// TwinCAT 3 PLC project PLC1
// ProgramVersion: 3.1.4022.2
// libraries:
//   Tc2_IoFunctions, * (Beckhoff Automation GmbH)
//   Tc2_ModbusRTU, * (Beckhoff Automation GmbH)
//   Tc2_ModbusSrv, * (Beckhoff Automation GmbH)
//   Tc2_Standard, * (Beckhoff Automation GmbH)
//   Tc2_System, * (Beckhoff Automation GmbH)
//   Tc3_Module, * (Beckhoff Automation GmbH)
//   Tc3_PLCopen_OpcUa, * (Beckhoff Automation GmbH)
// project tree:
//   DUTs/ ATV212.TcDUT, ATV212RegAddress.TcDUT, GrundfosMagna3.TcDUT (not stored), GrundfosRegAddress.TcDUT (not stored)
//   GVLs/ GVL.TcGVL, HWVar.TcGVL (not stored), Scale.TcGVL
//   / ModbusComm.TcTTO (not stored), PlcTask.TcTTO (not stored)
//   POUs/ BackgroundComm.TcPOU (not stored), IOConversion.TcPOU (not stored), MAIN.TcPOU (not stored), ModbusCommunication.TcPOU

// ---- DUTs/ATV212.TcDUT
TYPE ATV212 :
STRUCT
	fOutputFrequencyStatus	: REAL;
	fOutputCurrentStatus	: REAL;
	fOutputVoltageStatus	: REAL;
	fMotorSpeedStatus		: REAL;
END_STRUCT
END_TYPE

// ---- DUTs/ATV212RegAddress.TcDUT
{attribute 'qualified_only'}
TYPE ATV212RegAddress :
(
	listStart		:= 875,
	MotorSpeed		:= 875,
	OutputFrequency	:= 876,
	OutputCurrent	:= 877,
	OutputVoltage	:= 878,
	listEnd 		:= 879
) WORD := listStart;
END_TYPE

// ---- GVLs/GVL.TcGVL
{attribute 'qualified_only'}
VAR_GLOBAL
	{attribute 'OPC.UA.DA' := '1'}
	fTE         : ARRAY [1..19] OF REAL;
	{attribute 'OPC.UA.DA' := '1'}
    bHV AT %Q*  : ARRAY [1..11] OF BOOL;
	{attribute 'OPC.UA.DA' := '1'}
    bFan AT %Q*  : BOOL;
	{attribute 'OPC.UA.DA' := '1'}
    bST         : BOOL;
	{attribute 'OPC.UA.DA' := '1'}
	stP1		: GrundfosMagna3;
	{attribute 'OPC.UA.DA' := '1'}
	stP2		: GrundfosMagna3;
	{attribute 'OPC.UA.DA' := '1'}
	stFeeder	: ATV212;
	{attribute 'OPC.UA.DA' := '1'}
	bLoadTank1	: BOOL := TRUE;
	{attribute 'OPC.UA.DA' := '1'}
	bLoadTank2	: BOOL := TRUE;
	{attribute 'OPC.UA.DA' := '1'}
	bLoadTank3	: BOOL := TRUE;
END_VAR

// ---- GVLs/Scale.TcGVL
{attribute 'qualified_only'}
VAR_GLOBAL
	fGrundfosScale	: ARRAY [300..350] OF REAL := [
		0.001,		//Head                        
		0.1,		//VolumeFlow                 
		0.01,		//RelativePerformance        
		1.0,		//Speed                      
		0.1,		//Frequency                  
		1.0,		//DigitalInput               
		1.0,		//DigitalOutput              
		0.01,		//ActualSetpoint             
		0.1,		//MotorCurrent               
		0.1,		//DCLinkVoltage              
		0.1,		//MotorVoltage			    
		1.0,		//Power                      
		0.1,		//RemoteFlow                 
		0.001,		//InletPressure              
		0.001,		//RemotePressure             
		0.01,		//Level                      
		0.01,		//PowerElectronicTemp        
		0.01,		//MotorTemp                  
		0.01,		//RemoteTemp                 
		0.01,		//ElectronicTemp             
		0.01,		//PumpLiquidTemp             
		0.01,		//BearingTempDE			    
		0.01,		//BearingTempNDE             
		0.01,		//AuxSensorInput             
		1.0,		//SpecificEnergyConsumption  
		1.0,		//OperationTime                       
		1.0,		//TotalPoweredTime           
		0.1,		//Torque                     
		1.0,		//Energy                     
		1.0,		//NumberOfStarts             
		1.0,		//Reserved1                  
		0.01,		//RemoteTemp2                
		0.01,		//UserSetpoint               
		0.001,		//DiffPressure               
		0.001,		//OutletPressure             
		0.001,		//RemotePressure2            
		0.01,		//LoadPercent                
		1.0,		//PumpUnixRtc                
		0.1,		//MaxFlowLimit               
		0.01,		//RemoteDiffTemp             
		0.001,		//InletDiffPressure          
		0.001,		//OutletDiffPressure         
		0.001,		//RemoteDiffPressure         
		0.01,		//StorageTankLevel           
		0.01,		//AmbientTemp                
		1.0,		//HeatEnergyLifetime         
		1.0,		//HeatPower                  
		0.01,		//HeatDiffTemp               
		0.01,		//Volume                     
		1.0,		//HeatEnergyCounter2         
		0.01		//Volume2                    
	];
	fATV212Scale	: ARRAY [875..879] OF REAL := [
		1,			//Motor Speed                        
		0.01,		//Output frequency                
		0.01,		//Output current
		0.01		//Output votlage
	];
END_VAR

// ---- POUs/ModbusCommunication.TcPOU
PROGRAM ModbusCommunication
VAR
	aP1, aP2				: ARRAY [GrundfosRegAddress.listStart..GrundfosRegAddress.listEnd] OF WORD;
	aFeeder					: ARRAY [ATV212RegAddress.listStart..ATV212RegAddress.listEnd] OF WORD;
	nStep					: INT := 0;
END_VAR

VAR CONSTANT
	bP1Addr					: BYTE := 2;
	bP2Addr					: BYTE := 4;
	bFeederAddr				: BYTE := 5;
	wStartPumpCmd			: WORD := 16#0000;
	wStopPumpCmd			: WORD := 16#8000;
END_VAR

HWVar.ModbusMaster.ReadRegs(Execute := FALSE);
HWVar.ModbusMaster.WriteRegs(Execute := FALSE);
CASE nStep OF
	0:
		P1Read();
	1:
		P2Read();
	2:
		GrundfosDataConversion(arrReg:= aP1, pstGrundfosMagna3:= ADR(GVL.stP1));
		GrundfosDataConversion(arrReg:= aP2, pstGrundfosMagna3:= ADR(GVL.stP2));
		nStep := 3;
	3:	
		FeederRead();
	4:
		ATV212DataConversion(arrReg:=aFeeder, pstATV212:= ADR(GVL.stFeeder));
		nStep := 0;
END_CASE;

METHOD PRIVATE _P1Read : BOOL
VAR_STAT
	nRegisterAddress	: GrundfosRegAddress;
END_VAR
IF (NOT HWVar.ModbusMaster.BUSY) THEN
	HWVar.ModbusMaster.ReadRegs(
		UnitID := bP1Addr,
		Quantity := 1,
		MBAddr := nRegisterAddress,
		cbLength := 2,
		pMemoryAddr := ADR(aP1[nRegisterAddress]),
		Execute := TRUE,
		Timeout := T#5S,
		BUSY => ,
		Error =>
		);
	nRegisterAddress := nRegisterAddress+1;
	IF (nRegisterAddress = GrundfosRegAddress.listEnd + 1) THEN
		nStep := 1;
		nRegisterAddress :=  GrundfosRegAddress.listStart;
	END_IF
END_IF;
END_METHOD

METHOD PRIVATE _P2Read : BOOL
VAR_STAT
	nRegisterAddress	: GrundfosRegAddress;
END_VAR
IF (NOT HWVar.ModbusMaster.BUSY) THEN
	HWVar.ModbusMaster.ReadRegs(
		UnitID := bP2Addr,
		Quantity := 1,
		MBAddr := nRegisterAddress,
		cbLength := 2,
		pMemoryAddr := ADR((aP2[nRegisterAddress])),
		Execute := TRUE,
		Timeout := T#5S,
		BUSY => ,
		Error =>
		);
	nRegisterAddress := nRegisterAddress+1;
	IF (nRegisterAddress = GrundfosRegAddress.listEnd+1) THEN
		nStep := 2;
		nRegisterAddress :=  GrundfosRegAddress.listStart;
	END_IF
END_IF;
END_METHOD

METHOD ATV212DataConversion : BOOL
VAR_INPUT
	arrReg	: ARRAY [ATV212RegAddress.listStart..ATV212RegAddress.listEnd] OF WORD;
	pstATV212	: POINTER TO ATV212;
END_VAR

VAR
	iMemIndex: ATV212RegAddress;
	iRegIndex: ATV212RegAddress;
	a_MbRegValue	: ARRAY [300..350] OF REAL;
	dwMergedReg		: DWORD;
END_VAR
WHILE (iMemIndex <  ATV212RegAddress.listEnd AND iRegIndex < 879) DO
	IF (iRegIndex <> 875)
		AND (iRegIndex <> 876) 
		AND (iRegIndex <> 877)
		AND (iRegIndex <> 878) THEN
		a_MbRegValue[iRegIndex] := (arrReg[iMemIndex])*Scale.fATV212Scale[iRegIndex];
		iMemIndex := iMemIndex + 1;
		iRegIndex := iRegIndex + 1;
	ELSE
		dwMergedReg := SHL(WORD_TO_DWORD(arrReg[iMemIndex]),16) OR WORD_TO_DWORD(arrReg[iMemIndex+1]);
		a_MbRegValue[iRegIndex] := (dwMergedReg)*Scale.fATV212Scale[iRegIndex];
		iMemIndex := iMemIndex + 2;
		iRegIndex := iRegIndex + 1;
	END_IF
END_WHILE
MEMCPY(pstATV212, ADR(a_MbRegValue), SIZEOF(ATV212));
END_METHOD

METHOD FeederRead : BOOL
VAR_INPUT
END_VAR
IF (NOT HWVar.ModbusMaster.BUSY) THEN
	HWVar.ModbusMaster.ReadRegs(
		UnitID := bFeederAddr,
		Quantity := 4,
		MBAddr := 875,
		cbLength := SIZEOF(aFeeder),
		pMemoryAddr := ADR(aFeeder),
		Execute := TRUE,
		Timeout := T#5S,
		BUSY => ,
		Error =>
		);
		nStep := 4;
END_IF
END_METHOD

METHOD PUBLIC GrundfosDataConversion : BOOL
VAR_INPUT
	arrReg	: ARRAY [GrundfosRegAddress.listStart..GrundfosRegAddress.listEnd] OF WORD;
	pstGrundfosMagna3	: POINTER TO GrundfosMagna3;
END_VAR

VAR
	iMemIndex: GrundfosRegAddress;
	iRegIndex: GrundfosRegAddress;
	a_MbRegValue	: ARRAY [300..350] OF REAL;
	dwMergedReg		: DWORD;
END_VAR
WHILE (iMemIndex <  GrundfosRegAddress.listEnd AND iRegIndex < 351) DO
	IF (iRegIndex <> 311) 
		AND (iRegIndex <> 326)
		AND (iRegIndex <> 328) 
		AND (iRegIndex <> 331)
		AND (iRegIndex <> 323)
		AND (iRegIndex <> 342)
		AND (iRegIndex <> 351)
		AND (iRegIndex <> 353)
		AND (iRegIndex <> 356)
		AND (iRegIndex <> 358)
		AND (iRegIndex <> 360) THEN
		a_MbRegValue[iRegIndex] := (arrReg[iMemIndex])*Scale.fGrundfosScale[iRegIndex];
		iMemIndex := iMemIndex + 1;
		iRegIndex := iRegIndex + 1;
	ELSE
		dwMergedReg := SHL(WORD_TO_DWORD(arrReg[iMemIndex]),16) OR WORD_TO_DWORD(arrReg[iMemIndex+1]);
		a_MbRegValue[iRegIndex] := (dwMergedReg)*Scale.fGrundfosScale[iRegIndex];
		iMemIndex := iMemIndex + 2;
		iRegIndex := iRegIndex + 1;
	END_IF
END_WHILE
MEMCPY(pstGrundfosMagna3, ADR(a_MbRegValue), SIZEOF(GrundfosMagna3));
END_METHOD

METHOD PRIVATE P1Read : BOOL
VAR_STAT
	nRegisterAddress	: GrundfosRegAddress;
END_VAR
IF (NOT HWVar.ModbusMaster.BUSY) THEN
	HWVar.ModbusMaster.ReadRegs(
		UnitID := bP2Addr,
		Quantity := 62,
		MBAddr := 300,
		cbLength := SIZEOF(aP2),
		pMemoryAddr := ADR(aP2),
		Execute := TRUE,
		Timeout := T#5S,
		BUSY => ,
		Error =>
		);
		nStep := 1;
END_IF;
END_METHOD

METHOD PRIVATE P2Read : BOOL
VAR_STAT
	nRegisterAddress	: GrundfosRegAddress;
END_VAR
IF (NOT HWVar.ModbusMaster.BUSY) THEN
	HWVar.ModbusMaster.ReadRegs(
		UnitID := bP1Addr,
		Quantity := 62,
		MBAddr := 300,
		cbLength := SIZEOF(aP1),
		pMemoryAddr := ADR(aP1),
		Execute := TRUE,
		Timeout := T#5S,
		BUSY => ,
		Error =>
		);
		nStep := 2;
END_IF;
END_METHOD

ACTION SC01Read:
nStep := 3;
END_ACTION

END_PROGRAM
